FUNCTION_BLOCK PUBLISH_6 (* Generic publish (6 SD, 0 RD); instantiated from GEN_PUBLISH *)
  (* Standard: 61499-2 *)
  (* Version 0.1, 2026-09-28, Project contributors, AAU Smart Production Lab *)
  PACKAGE iec61499::net;
  {SET_ATTRIBUTE(eclipse4diac::core::GenericClassName, 'GEN_PUBLISH')}
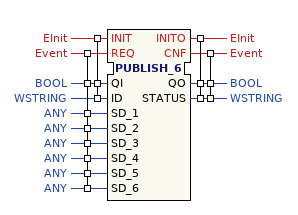
  EVENT_INPUT
    INIT : EInit WITH QI, ID;
    REQ WITH QI, SD_1, SD_2, SD_3, SD_4, SD_5, SD_6;
  END_EVENT
  EVENT_OUTPUT
    INITO : EInit WITH QO, STATUS;
    CNF WITH QO, STATUS;
  END_EVENT
  VAR_INPUT
    QI : BOOL;
    ID : WSTRING;
    SD_1 : ANY;
    SD_2 : ANY;
    SD_3 : ANY;
    SD_4 : ANY;
    SD_5 : ANY;
    SD_6 : ANY;
  END_VAR
  VAR_OUTPUT
    QO : BOOL;
    STATUS : WSTRING;
  END_VAR
END_FUNCTION_BLOCK
